// TIA Portal V21 export
VAR_GLOBAL   // PLC tag table "Default tag table"
   "REC DOOR1 PRESSURE" AT %QW150 : Int;
   "REC DOOR2 PRESSURE" AT %QW152 : Int;
   "REC CHAMBER PRESSURE" AT %QW154 : Int;
   "REC JACKET PRESSURE" AT %QW156 : Int;
   "REC DRUM SPEED" AT %QW158 : Int;
   "PRINT START" AT %M0.0 : Bool;
   TRIGGER AT %M0.1 : Bool;
   LENGTH AT %MW2 : Int;
   "NOT" AT %M0.2 : Bool;
   HIT AT %M0.3 : Bool;
   "START PV" AT %M0.4 : Bool;
   Clock_Byte AT %MB500 : Byte;
   Clock_10Hz AT %M500.0 : Bool;
   Clock_5Hz AT %M500.1 : Bool;
   "Clock_2.5Hz" AT %M500.2 : Bool;
   Clock_2Hz AT %M500.3 : Bool;
   "Clock_1.25Hz" AT %M500.4 : Bool;
   Clock_1Hz AT %M500.5 : Bool;
   "Clock_0.625Hz" AT %M500.6 : Bool;
   "Clock_0.5Hz" AT %M500.7 : Bool;
   System_Byte AT %MB1 : Byte;
   FirstScan AT %M1.0 : Bool;
   DiagStatusUpdate AT %M1.1 : Bool;
   AlwaysTRUE AT %M1.2 : Bool;
   AlwaysFALSE AT %M1.3 : Bool;
   AHJGSJH AT %MB4 : Byte;
   JGJH AT %MB5 : Byte;
   GET_DAY AT %MB180 : Byte;
   GET_MONTH AT %MB181 : Byte;
   GET_YEAR AT %MB182 : Byte;
   DAY AT %MW32 : Int;
   MONTH AT %MW44 : Int;
   YEAR AT %MW10 : Int;
   GET_HOUR AT %MB183 : Byte;
   GET_MINUTE AT %MB184 : Byte;
   GET_SECOND AT %MB185 : Byte;
   HOUR AT %MW40 : Int;
   MINUTE AT %MW42 : Int;
   SECOND AT %MW12 : Int;
   "NILESH BHAU" AT %MB6 : Byte;
   GET_CONTROL_TEMP AT %MD1400 : Real;
   "SP_CONTROL TEMP" AT %MD60 : Real;
   GET_CONVEYOR_SPEED AT %MD1404 : Real;
   SP_CONVEYOR_SPEED AT %MD64 : Real;
   "DRY ZONE REAL" AT %MD16 : Real;
   "GET_CONVEYOR ON TEMP" AT %MD1408 : Real;
   SP_CONVEYOR_ON_TEMP AT %MD68 : Real;
   "GET_CONVEYOR OFF TEMP" AT %MD1412 : Real;
   SP_CONVEYOR_OFF_TEMP AT %MD72 : Real;
   GET_DZ_PV AT %MD1416 : Real;
   DZ_PV AT %MD20 : Real;
   GET_MHZ_PV AT %MD1420 : Real;
   MHZ_PV AT %MD76 : Real;
   GET_STR_IN_PV AT %MD1424 : Real;
   STR_IN_PV AT %MD24 : Real;
   GET_STR_OUT_PV AT %MD1428 : Real;
   STR_OUT_PV AT %MD80 : Real;
   GET_CLZ_UP_PV AT %MD1432 : Real;
   CLZ_UP_PV AT %MD84 : Real;
   GET_CLZ_DWN_PV AT %MD1436 : Real;
   CLZ_DWN_PV AT %MD28 : Real;
   "GET_CONVEYOR SPEED_PV" AT %MD1440 : Real;
   "CONVEYOR SPEED_PV" AT %MD36 : Real;
   KJAHKJH AT %MD46 : Real;
   GET_MODE AT %MB197 : Byte;
   MODE AT %MW14 : Int;
   GET_PROCESS_HOUR AT %MB198 : Byte;
   PROCESS_HOUR AT %MW50 : Int;
   GET_PROCESS_MINUTE AT %MB199 : Byte;
   PROCESS_MINUTE AT %MW52 : Int;
   GET_PROCESS_SEC AT %MB200 : Byte;
   PROCESS_SEC AT %MW54 : Int;
   AL1 AT %M115.0 : Bool;
   "AL EMG STOP" AT %M115.1 : Bool;
   "AL DRUM TRIP" AT %M115.2 : Bool;
   "AL VACUUM TRIP" AT %M115.3 : Bool;
   "AL CRC TRIP" AT %M115.4 : Bool;
   AL6 AT %M115.5 : Bool;
   AL7 AT %M115.6 : Bool;
   AL8 AT %M115.7 : Bool;
   AL9 AT %M114.0 : Bool;
   AL10 AT %M114.1 : Bool;
   AL11 AT %M114.2 : Bool;
   AL12 AT %M114.3 : Bool;
   "AL JACKET RTD FAIL" AT %M114.4 : Bool;
   "AL CHAM RTD FAIL" AT %M114.5 : Bool;
   "AL AIR FAIL" AT %M114.6 : Bool;
   AL16 AT %M114.7 : Bool;
   AL1_1 AT %M118.0 : Bool;
   AL1_2 AT %M118.1 : Bool;
   AL1_3 AT %M118.2 : Bool;
   "AL JACKET PRESS FAIL" AT %M118.3 : Bool;
   "AL DOOR1 PRESS FAIL" AT %M118.4 : Bool;
   "AL DOOR2 PRESS FAIL" AT %M118.5 : Bool;
   "AL CHAM PRESS FAIL" AT %M118.6 : Bool;
   AL1_8 AT %M118.7 : Bool;
   "AL DOOR1 CL LMT FAIL" AT %M117.0 : Bool;
   AL2_10 AT %M117.1 : Bool;
   AL2_11 AT %M117.2 : Bool;
   AL2_12 AT %M117.3 : Bool;
   "AL DOOR2 CL LMT FAIL" AT %M117.4 : Bool;
   AL2_14 AT %M117.5 : Bool;
   AL2_15 AT %M117.6 : Bool;
   AL2_16 AT %M117.7 : Bool;
   "REQ AL1" AT %M0.5 : Bool;
   "AL1 TRIG" AT %M0.6 : Bool;
   "REQ AL3" AT %M0.7 : Bool;
   "AL3 TRIG" AT %M7.0 : Bool;
   "REQ AL4" AT %M7.1 : Bool;
   "AL4 TRIG" AT %M7.2 : Bool;
   "AL5 TRIG" AT %M7.3 : Bool;
   "REQ AL5" AT %M7.4 : Bool;
   "AL6 TRIG" AT %M7.5 : Bool;
   "REQ AL6" AT %M7.6 : Bool;
   "AL7 TRIG" AT %M7.7 : Bool;
   "REQ AL7" AT %M56.0 : Bool;
   "AL8 TRIG" AT %M56.1 : Bool;
   "REQ AL8" AT %M56.2 : Bool;
   "AL11 TRIG" AT %M56.3 : Bool;
   "REQ AL11" AT %M56.4 : Bool;
   "AL12 TRIG" AT %M56.5 : Bool;
   "REQ AL12" AT %M56.6 : Bool;
   "AL14 TRIG" AT %M56.7 : Bool;
   "REQ AL14" AT %M57.0 : Bool;
   "AL1_1 TRIG" AT %M57.1 : Bool;
   "REQ AL1_1" AT %M57.2 : Bool;
   "AL1_3 TRIG" AT %M57.3 : Bool;
   "REQ AL1_3" AT %M57.4 : Bool;
   "AL1_5 TRIG" AT %M57.5 : Bool;
   "REQ AL1_5" AT %M57.6 : Bool;
   "AL1_6 TRIG" AT %M57.7 : Bool;
   "REQ AL1_6" AT %M58.0 : Bool;
   "AL1_7 TRIG" AT %M58.1 : Bool;
   "REQ AL1_7" AT %M58.2 : Bool;
   "AL1_8 TRIG" AT %M58.3 : Bool;
   "REQ AL1_8" AT %M58.4 : Bool;
   "AL2_9 TRIG" AT %M58.5 : Bool;
   "REQ AL2_9" AT %M58.6 : Bool;
   "AL2_14 TRIG" AT %M58.7 : Bool;
   "REQ AL2_14" AT %M59.0 : Bool;
   "EMG SEL BIT" AT %M8.0 : Bool;
   "PHASE FAIL SEL BIT" AT %M8.1 : Bool;
   "COVEYOR SEL BIT" AT %M8.2 : Bool;
   "HEATER SEL BIT" AT %M8.3 : Bool;
   "TEMP SEL BIT" AT %M8.4 : Bool;
   "DRY ZONE SEL BIT" AT %M8.5 : Bool;
   "COOL ZONE SEL BIT" AT %M8.6 : Bool;
   "STR ZONE BIT" AT %M8.7 : Bool;
   "VAPOR TRIP SEL BIT" AT %M9.0 : Bool;
   "TURBINE TRIP SEL BIT" AT %M9.1 : Bool;
   "VAPOR SUPPLY SEL BIT" AT %M9.2 : Bool;
   "CONV OVER SEL BIT" AT %M9.3 : Bool;
   "LAF FAIL SEL BIT" AT %M9.4 : Bool;
   "GET_SHUDOWN BUFF" AT %MW1444 : Int;
   "SHUDOWN BUFF" AT %MW34 : Int;
   SHUT AT %M9.5 : Bool;
   "REQ SHUT" AT %M9.6 : Bool;
   LAST AT %MB1446 : Byte;
   "LAST TRIG" AT %M9.7 : Bool;
   OVER AT %M59.1 : Bool;
   "P OVER" AT %M59.2 : Bool;
   "PRINT STOP" AT %M59.3 : Bool;
   "PRINT STOP TRIG" AT %M59.4 : Bool;
   "HEAT UP 1 ON" AT %M59.5 : Bool;
   "HEAT UP 2 ON" AT %M59.6 : Bool;
   "HEAT UP 3 ON" AT %M59.7 : Bool;
   "HEAT UP 4 ON" AT %M88.0 : Bool;
   "CONV TEMP ON" AT %M88.1 : Bool;
   "V HIGH PRESS" AT %M151.0 : Bool;
   "AL DOOR2 OP LMT FAIL" AT %M151.1 : Bool;
   "AL DOOR1 OP LMT FAIL" AT %M151.2 : Bool;
   "AL STER_TIME_STOP" AT %M700.0 : Bool;
   "AL TURB SUP FAIL" AT %M151.4 : Bool;
   "AL STER_HOLD TIME RESET" AT %M151.5 : Bool;
   "AL HEATER SUP FAIL" AT %M151.6 : Bool;
   "AL_JACKET HEATING FAIL" AT %M151.7 : Bool;
   "AL_STER_HOLD HEATING FAIL" AT %M150.0 : Bool;
   AL_TOO_LATE_VACUUM AT %M150.1 : Bool;
   "AL BOILER WATER LOW" AT %M150.2 : Bool;
   "AL_DOOR1 SAFETY SENSOR FAIL" AT %M150.3 : Bool;
   "AL PHASE FAIL" AT %M150.4 : Bool;
   "1ML OK" AT %M88.2 : Bool;
   "2ML OK" AT %M88.3 : Bool;
   "3ML OK" AT %M88.4 : Bool;
   "5ML OK" AT %M88.5 : Bool;
   "10ML OK" AT %M88.6 : Bool;
   "HOOTER RESET BIT" AT %M88.7 : Bool;
   "CON ANNI" AT %M89.0 : Bool;
   "MANUAL INFEED" AT %M89.1 : Bool;
   "VPR ANN" AT %M89.2 : Bool;
   "LAF ANN" AT %M89.3 : Bool;
   "100ML OK" AT %M89.4 : Bool;
   "TURBINE SUP SEL BIT" AT %M89.5 : Bool;
   "AL VACUUM BREAK FAIL" AT %M150.6 : Bool;
   "AL DOOR PRECOND FAIL" AT %M150.7 : Bool;
   "AL JACKET PRESSURE HH" AT %M153.0 : Bool;
   BL1 AT %MW90 : Int;
   "AL DRY ZONE HIGH" AT %M153.2 : Bool;
   RESET AT %M89.6 : Bool;
   "LAF ON" AT %M89.7 : Bool;
   OFF AT %M92.0 : Bool;
   "VPR ON" AT %M92.1 : Bool;
   OFF1 AT %M92.2 : Bool;
   "TURB ON" AT %M92.3 : Bool;
   OFF2 AT %M92.4 : Bool;
   "HEAT ON" AT %M92.5 : Bool;
   OFF3 AT %M92.6 : Bool;
   "CONV ON" AT %M92.7 : Bool;
   "OFF 4" AT %M93.0 : Bool;
   "DOWNLOAD RC" AT %M93.1 : Bool;
   "AL HOT PRS LOW" AT %M153.1 : Bool;
   "AL COOL PRS HIGH" AT %M153.3 : Bool;
   Tag_1 AT %M153.4 : Bool;
   "AL CONV OVER" AT %M153.5 : Bool;
   "AL LAF PRESS SWS" AT %M153.6 : Bool;
   "HEATER 2" AT %M93.2 : Bool;
   OFFF AT %M93.3 : Bool;
   "HEATER 3" AT %M93.4 : Bool;
   OFFF1 AT %M93.5 : Bool;
   "HEATER 4" AT %M93.6 : Bool;
   OFFF44 AT %M93.7 : Bool;
   Tag_3 AT %M153.7 : Bool;
   Tag_4 AT %M152.0 : Bool;
   "CONVEYOR TRIP SEL BIT" AT %M110.0 : Bool;
   OFFFFFF AT %M94.0 : Bool;
   "PRINT SPEED" AT %MD96 : Real;
   TURBINE2 AT %M94.1 : Bool;
   OK AT %M94.2 : Bool;
   RESETC1 AT %M94.3 : Bool;
   POPUP AT %M152.1 : Bool;
   RESETC3 AT %M94.4 : Bool;
   RESETC4 AT %M94.5 : Bool;
   RESETC5 AT %M94.6 : Bool;
   RESETC6 AT %M94.7 : Bool;
   RESETC7 AT %M95.0 : Bool;
   RESETC8 AT %M95.1 : Bool;
   RESETC9 AT %M95.2 : Bool;
   RESETC10 AT %M95.3 : Bool;
   RESETC11 AT %M95.4 : Bool;
   RESETT5 AT %M95.5 : Bool;
   RESETC12 AT %M95.6 : Bool;
   RESETT6 AT %M95.7 : Bool;
   RESETC13 AT %M100.0 : Bool;
   RESETT7 AT %M100.1 : Bool;
   RESETC14 AT %M100.2 : Bool;
   RESETT8 AT %M100.3 : Bool;
   RESETC15 AT %M100.4 : Bool;
   RESETC16 AT %M100.5 : Bool;
   RESETC17 AT %M100.6 : Bool;
   RESETC18 AT %M100.7 : Bool;
   RESETT12 AT %M101.0 : Bool;
   RESETC19 AT %M101.1 : Bool;
   RESETC20 AT %M101.2 : Bool;
   RESETC21 AT %M101.3 : Bool;
   RESETC22 AT %M101.4 : Bool;
   RESETT16 AT %M101.5 : Bool;
   RESETC23 AT %M101.6 : Bool;
   RESETC24 AT %M101.7 : Bool;
   RESETC25 AT %M102.0 : Bool;
   RESETC26 AT %M102.1 : Bool;
   RESETC27 AT %M102.2 : Bool;
   RESETT21 AT %M102.3 : Bool;
   RESETC28 AT %M102.4 : Bool;
   RESETT22 AT %M102.5 : Bool;
   RESETC29 AT %M102.6 : Bool;
   RESETT23 AT %M102.7 : Bool;
   RESETC30 AT %M103.0 : Bool;
   "DRUM MOTOR BIT" AT %M103.1 : Bool;
   "EXH ON" AT %M103.2 : Bool;
   RESETC32 AT %M103.3 : Bool;
   "CONTROL CHMB" AT %M103.4 : Bool;
   "STERILE TEMP ON" AT %MD104 : Real;
   "PWD TEMP ON" AT %MD120 : Real;
   resetc33 AT %M103.5 : Bool;
   "vaccum ok" AT %M103.6 : Bool;
   trigger2 AT %M103.7 : Bool;
   "VCC DIFF" AT %MD124 : Real;
   LENGTH2 AT %MW108 : Int;
   "CYCLE END" AT %M110.1 : Bool;
   ERROR AT %M110.2 : Bool;
   "RESET HPHV VCC" AT %M110.3 : Bool;
   "RESETBOW VCC" AT %M110.4 : Bool;
   okkk AT %M110.5 : Bool;
   "one shot" AT %M110.6 : Bool;
   "jack out set" AT %M110.7 : Bool;
   resetct3 AT %M111.0 : Bool;
   resetct4 AT %M111.1 : Bool;
   "hphv ok" AT %M111.2 : Bool;
   "bowie ok" AT %M111.3 : Bool;
   "std ok" AT %M111.4 : Bool;
   sterileok AT %M111.5 : Bool;
   "TEST BIT" AT %M111.6 : Bool;
   "TEST BIT2" AT %M111.7 : Bool;
   "CLOSURE ON" AT %M112.0 : Bool;
   "CLOSE START" AT %M112.1 : Bool;
   "DEL LENGTH" AT %MW128 : Int;
   "RESET C5" AT %M112.2 : Bool;
   sip_ok AT %M112.3 : Bool;
   "sip ok1" AT %M112.4 : Bool;
   PULSE1 AT %M112.5 : Bool;
   PULSE2 AT %M112.6 : Bool;
   pulse3 AT %M112.7 : Bool;
   PP1 AT %M113.0 : Bool;
   PP2 AT %M113.1 : Bool;
   PP3 AT %M113.2 : Bool;
   PP4 AT %M113.3 : Bool;
   PP5 AT %M113.4 : Bool;
   pp6 AT %M113.5 : Bool;
   RESETCOUNT6 AT %M113.6 : Bool;
   RESETCOUNT7 AT %M113.7 : Bool;
   "VACCUM LEAK DIFF" AT %MD130 : Real;
   PULSE4 AT %M116.0 : Bool;
   PULSE5 AT %M116.1 : Bool;
   PULSE6 AT %M116.2 : Bool;
   PULSE7 AT %M116.3 : Bool;
   PULSE8 AT %M116.4 : Bool;
   PULSE9 AT %M116.5 : Bool;
   PULSE10 AT %M116.6 : Bool;
   PULSE11 AT %M116.7 : Bool;
   PULSE12 AT %M119.0 : Bool;
   PULSE13 AT %M119.1 : Bool;
   pulse14 AT %M119.2 : Bool;
   pulse15 AT %M119.3 : Bool;
   "STD1 SELECT" AT %M119.4 : Bool;
   "STD2 SELECT" AT %M119.5 : Bool;
   PULSE16 AT %M119.6 : Bool;
   PULSE17 AT %M119.7 : Bool;
   PULSE18 AT %M134.0 : Bool;
   PULSE19 AT %M134.1 : Bool;
   PULSE20 AT %M134.2 : Bool;
   pulse21 AT %M134.3 : Bool;
   "END PRINT OK" AT %M134.4 : Bool;
   PULSE22 AT %M134.5 : Bool;
   pulse23 AT %M134.6 : Bool;
   pulse24 AT %M134.7 : Bool;
   pulse25 AT %M135.0 : Bool;
   pulse26 AT %M135.1 : Bool;
   pulse27 AT %M135.2 : Bool;
   pulse28 AT %M135.3 : Bool;
   pulse29 AT %M135.4 : Bool;
   pulse30 AT %M135.5 : Bool;
   pulse31 AT %M135.6 : Bool;
   pulse32 AT %M135.7 : Bool;
   pulse33 AT %M136.0 : Bool;
   pulse34 AT %M136.1 : Bool;
   pulse35 AT %M136.2 : Bool;
   pulse36 AT %M136.3 : Bool;
   pulse37 AT %M136.4 : Bool;
   pulse38 AT %M136.5 : Bool;
   pulse39 AT %M136.6 : Bool;
   pulse40 AT %M136.7 : Bool;
   "start process" AT %M137.0 : Bool;
   PULSE41 AT %M137.1 : Bool;
   "START PROCES2" AT %M137.2 : Bool;
   PULSE42 AT %M137.3 : Bool;
   pulse43 AT %M137.4 : Bool;
   PULSE44 AT %M137.5 : Bool;
   PULSE45 AT %M137.6 : Bool;
   PULSE46 AT %M137.7 : Bool;
   PULSE47 AT %M138.0 : Bool;
   PULSE48 AT %M138.1 : Bool;
   PULSE49 AT %M138.2 : Bool;
   "hooter reset" AT %M138.3 : Bool;
   "RESET DOOR1" AT %M138.4 : Bool;
   "RESET DOOR2" AT %M138.5 : Bool;
   "STD3 SELECT" AT %M138.6 : Bool;
   "STD4 SELECT" AT %M138.7 : Bool;
   "STD5 SELECT" AT %M139.0 : Bool;
   "STD6 SELECT" AT %M139.1 : Bool;
   "STD7 SELECT" AT %M139.2 : Bool;
   "STD8 SELECT" AT %M139.3 : Bool;
   "STD9 SELECT" AT %M139.4 : Bool;
   "VACCUM FAIL" AT %M139.5 : Bool;
   "hold start" AT %M139.6 : Bool;
   RESETT169 AT %M139.7 : Bool;
   RESET_C8 AT %M140.0 : Bool;
   RESETT171 AT %M140.1 : Bool;
   RESETC_9 AT %M140.2 : Bool;
   RESETT174 AT %M140.3 : Bool;
   RESET_C10 AT %M140.4 : Bool;
   RESETT177 AT %M140.5 : Bool;
   RESET_C11 AT %M140.6 : Bool;
   RESETT179 AT %M140.7 : Bool;
   RESET_C12 AT %M141.0 : Bool;
   RESETT184 AT %M141.1 : Bool;
   RESET_C13 AT %M141.2 : Bool;
   RESETT185 AT %M141.3 : Bool;
   RESET_C14 AT %M141.4 : Bool;
   RESET_C15 AT %M141.5 : Bool;
   "RESET C16" AT %M141.6 : Bool;
   "RESET C17" AT %M141.7 : Bool;
   "reset c18" AT %M142.0 : Bool;
   RESET_C19 AT %M142.1 : Bool;
   "STANDARD DONE" AT %M142.2 : Bool;
   "HPHV DONE" AT %M142.3 : Bool;
   "BOW DONE" AT %M142.4 : Bool;
   "VACUUM DONE" AT %M142.5 : Bool;
   PULSE50 AT %M142.6 : Bool;
   "RESET C7" AT %M142.7 : Bool;
   pulse51 AT %M143.0 : Bool;
   pulse52 AT %M143.1 : Bool;
   Tag_2 AT %M151.3 : Bool;
   "VLT OG" AT %M143.2 : Bool;
   "VLT EX" AT %M143.3 : Bool;
   AMP_VLT AT %M143.4 : Bool;
   "CYCLE STOP PRESS" AT %M143.5 : Bool;
   PULSE53 AT %M143.6 : Bool;
   "STER HEAT AGAIN" AT %M143.7 : Bool;
   "STER HEAT FAIL" AT %M144.0 : Bool;
   PULSE54 AT %M144.1 : Bool;
   PULSE55 AT %M144.2 : Bool;
   reset_c20 AT %M144.3 : Bool;
   PULSE60 AT %M144.4 : Bool;
   PULSE61 AT %M144.5 : Bool;
   PULSE62 AT %M144.6 : Bool;
   PULSE56 AT %M144.7 : Bool;
   "AL_DOOR2 SAFETY SENSOR FAIL" AT %M150.5 : Bool;
   "BOILER WATER INLET VAL" AT %Q3.7 : Bool;
END_VAR
